// TwinCAT 3 PLC project FRANKA
// ProgramVersion: 3.1.4023.0
// libraries:
//   Tc2_Database, * (Beckhoff Automation GmbH)
//   Tc2_ModbusRTU, * (Beckhoff Automation GmbH)
//   Tc2_ModbusSrv, * (Beckhoff Automation GmbH)
//   Tc2_Standard, * (Beckhoff Automation GmbH)
//   Tc2_System, * (Beckhoff Automation GmbH)
//   Tc2_Utilities, * (Beckhoff Automation GmbH)
//   Tc3_Database, * (Beckhoff Automation GmbH)
//   Tc3_EventLogger, * (Beckhoff Automation GmbH)
//   Tc3_Module, * (Beckhoff Automation GmbH)
//   VisuSymbols,3.5.10.0,System
// project tree:
//   DUTs/ MS.TcTLEO, PLC_Data.TcDUT, ST_Table.TcDUT, DB_Columns.TcDUT, Visu_Data.TcDUT
//   / GlobalTextList.TcGTLO, PlcTask.TcTTO, Visualisierungsmanager.TcVMO (not stored)
//   GVLs/ GVL.TcGVL, GVL_IO.TcGVL, GVL_Persistent.TcGVL
//   POUs/ FB_Blinker.TcPOU, Initialize_Measurement_Values.TcPOU, MAIN.TcPOU, FB_NewTable.TcPOU, FB_DB_Write2.TcPOU, shutdown.TcPOU
//   VISUs/ Visualization.TcVIS
// real-time tasks:
//   TASK PlcTask: cycle T#10ms, priority 20, ADS port 350
//   TASK PlcTask1: cycle T#10ms, priority 21, ADS port 351
// I/O:
//   DEVICE Gerät 1 (EtherCAT Automation Protocol) (disabled), AmsNetId 192.168.26.100.2.1
//   DEVICE Gerät 3 (EtherCAT), AmsNetId 192.168.26.100.4.1
//     Klemme 1 (EK1100) [EK1100 EtherCAT-Koppler (2A E-Bus)]
//       Klemme 2 (EL2008) [EL2008 8K. Dig. Ausgang 24V, 0.5A]
//       Klemme 3 (EL2008) [EL2008 8K. Dig. Ausgang 24V, 0.5A]
//       Klemme 4 (EL1008) [EL1008 8K. Dig. Eingang 24V, 3ms]
//       Klemme 5 (EL2024) [EL2024 4K. Dig. Ausgang 24V, 2A]
//       Klemme 6 (EL9011) [EL9011 Endklemme]
// variable links:
//   FRANKA/FRANKA Instance <-> Device 3 (EtherCAT)/Term 1 (EK1100)/Term 2 (EL2008)
//     PlcTask Outputs/GVL.LED1 <-> Channel 4/Output
//     PlcTask Outputs/GVL.LED2 <-> Channel 1/Output
//     PlcTask Outputs/GVL.LED3 <-> Channel 7/Output
//     PlcTask Outputs/GVL.LED4 <-> Channel 6/Output
//     PlcTask Outputs/GVL.LED5 <-> Channel 8/Output
//     PlcTask Outputs/GVL.LED6 <-> Channel 3/Output
//     PlcTask Outputs/GVL.LED7 <-> Channel 5/Output
//     PlcTask Outputs/GVL.LED8 <-> Channel 2/Output
//   FRANKA/FRANKA Instance <-> Device 3 (EtherCAT)/Term 1 (EK1100)/Term 3 (EL2008)
//     PlcTask Outputs/GVL.Schalterlichtgrun <-> Channel 3/Output
//     PlcTask Outputs/GVL.Schalterlichtrot <-> Channel 1/Output
//     PlcTask Outputs/GVL.Schalterlichtweis <-> Channel 4/Output
//     PlcTask Outputs/GVL.schalterspannung <-> Channel 2/Output
//   FRANKA/FRANKA Instance <-> Device 3 (EtherCAT)/Term 1 (EK1100)/Term 4 (EL1008)
//     PlcTask Inputs/GVL.Grau_Schalter <-> Channel 1/Input
//     PlcTask Inputs/GVL.Start_Schalter <-> Channel 2/Input
//     PlcTask Inputs/GVL.Stop_Schalter <-> Channel 3/Input

CONFIGURATION FRANKA
    RESOURCE PLC ON TwinCAT3
        TASK PlcTask(INTERVAL := T#10ms, PRIORITY := 20);
        PROGRAM MAIN WITH PlcTask : MAIN;
    END_RESOURCE
END_CONFIGURATION

// ---- DUTs/MS.TcTLEO
{attribute 'qualified_only'}
{attribute 'strict'}
TYPE MS :
(
	Init_delay,
	Initialization,
	Start,
	Restart,
	NewTable_DB,
	Write_DB,
	FRANKA_Pick_and_place_PCB,
	FRANKA_Measure,
	LED_confirmation,
	FRANKA_Place_PCB,
	DB_Write,
	Measurement_counter,
	Reset,
	FRANKA_ERROR,
	measurebackup,
	Wait
	
);
END_TYPE

// ---- DUTs/PLC_Data.TcDUT
TYPE PLC_Data :
STRUCT
	PCB_ID			: 	INT;
	PCB_no_defects	:	STRING(50);
	Measurement_ID	: 	ARRAY [1..6] OF INT;
	TimeStamp		: 	ARRAY [1..6] OF DT;
	MeasureInTol	: 	ARRAY [1..6] OF STRING(50);
	Measure_Type	: 	ARRAY [1..6] OF STRING(50);
	Measure_Result	: 	ARRAY [1..6] OF REAL;
	Measure_Reference: 	ARRAY [1..6] OF REAL;
	Measure_Tolerance: 	ARRAY [1..6] OF REAL;

END_STRUCT
END_TYPE

// ---- DUTs/ST_Table.TcDUT
TYPE ST_Table :
STRUCT
sName: STRING(50);
sProperty: STRING;
nLength: UDINT;
eType: E_ColumnType;
END_STRUCT
END_TYPE

// ---- DUTs/DB_Columns.TcDUT
TYPE DB_Columns :
STRUCT
	PCB_Batch_ID: INT;
	PCB_ID: 		INT;
	Measurement_ID: INT;
	TimeStamp: 		DT;
	FreeFromDefects: STRING(50);
	Measure_Type: STRING(50);
	Measure_Result: REAL;
	Measure_Reference: REAL;
	Measure_Tolerance: REAL;	
END_STRUCT
END_TYPE

// ---- DUTs/Visu_Data.TcDUT
TYPE Visu_Data :
STRUCT
	PCB_Batch_ID	: 		INT;	
	PCB_ID			: 		INT;
	PCB_no_defects	:		STRING(50);
	Measure1InTol	: 		STRING(50);
	Measure2InTol	: 		STRING(50);
	Measure3InTol	: 		STRING(50);		
END_STRUCT
END_TYPE

// ---- GVLs/GVL.TcGVL
 {attribute 'qualified_only'}
VAR_GLOBAL
//Preset before program
	pcb_n			: INT;
	measure_n 		: INT;
	pcb_max			: INT;
	measure_max		: INT;

// MS Access Table Setting	
	ActiveTable		: STRING;
	
	
// fill during program
    Data: DB_Columns; // Data for MS Access Database
	PLC_Data: ARRAY [1..8] OF PLC_Data;// Data Saved in PLC
	Visu_Data: ARRAY [1..8] OF Visu_Data; // Visu Data
	

// DB_Writting
	Writing_finished: BOOL;
	write_state: INT;
	
// I/O Configuration
	
	LED1	AT%Q*:	BOOL;
	LED2	AT%Q*:	BOOL;
	LED3	AT%Q*:	BOOL;
	LED4	AT%Q*:	BOOL;
	LED5	AT%Q*:	BOOL;
	LED6	AT%Q*:	BOOL;
	LED7	AT%Q*:	BOOL;
	LED8	AT%Q*:	BOOL;
	
	Schalterlichtrot 	AT%Q*:	BOOL;
	Schalterlichtweis 	AT%Q*:	BOOL;
	Schalterlichtgrun 	AT%Q*:	BOOL;
	schalterspannung 	AT%Q*:	BOOL;
	
	Start_Schalter	AT%I*:	BOOL;
	Stop_Schalter	AT%I*:	BOOL;
	Grau_Schalter	AT%I*:	BOOL;
	
// Modbus Variabeln
	mb_Input_Coils      : ARRAY [0..255] OF BOOL;
	mb_Output_Coils     : ARRAY [0..255] OF BOOL;
	mb_Input_Registers  : ARRAY [0..255] OF WORD;
	mb_Output_Registers : ARRAY [0..255] OF WORD;

// Variables Measurement
	
sMeas_type	:	STRING;	// Measurement type first define measurement type then start
						// CSQ | CSD | CSR | CPQ | CPD | CPR | CPG | LSQ |LSD | LSR |
						// LPQ | LPD | LPR | LPG | ZTH | YTH | RX | GB | DCR |
bMeas_start	:	BOOL;	// start mearuement
rMeas_01	: 	REAL;	// Measurement result 1
rMeas_02	: 	REAL;	// Measurement result 2
bMeas_ready	:	BOOL;	// Measurement finished
bMeas_error	:	BOOL;	// Error flag
sMeas_errormsg:	STRING;	// Error Message String
bkill_proc	:	BOOL;	// Terminate Python Script

// Blocky start

        bStartBlockly 	: BOOL 		:= TRUE;
		sDeskUsername	: STRING 	:='Benjamin';
		sDeskPassword	: STRING	:='Benjamin';

// Init Measurement settings
Measurement_Init : BOOL;


END_VAR

// ---- GVLs/GVL_IO.TcGVL
{attribute 'qualified_only'}
VAR_GLOBAL
	// FRANKA OUTPUT Coils
	
	FRANKA_Marker0			:	REFERENCE TO BOOL;
	FRANKA_home1			:	REFERENCE TO BOOL;
	PCB_Marker2				: 	REFERENCE TO BOOL;
	FRANKA_MPoint_reached3	:	REFERENCE TO BOOL;
	FRANKA_Measurement_finished4: REFERENCE TO BOOL;
	FRANKA_PCB_Picked5		:	REFERENCE TO BOOL;
	FRANKA_PCB_Placed6		:	REFERENCE TO BOOL;
	FRANKA_ready_to_start	:	REFERENCE TO BOOL;

	// FRANKA INPUT Coils
	PLC_Measure_Finished0	: 	REFERENCE TO BOOL;
	PLC_confirm_PCB_placement1: 	REFERENCE TO BOOL;
	PLC_Start_trigger		:	REFERENCE TO BOOL;
	
END_VAR

// ---- GVLs/GVL_Persistent.TcGVL
{attribute 'qualified_only'}
VAR_GLOBAL PERSISTENT
		PCB_Batch_ID			: INT;


END_VAR

// ---- POUs/MAIN.TcPOU
PROGRAM MAIN
VAR




state : MS;

NewTable 	: FB_NewTable;
WriteDB		: FB_DB_Write;



// current file time

		fbSystemTime    : GETSYSTEMTIME;
        timeAsFileTime  : T_FILETIME;
        timeAsDT        : DT;
// Measurement trigger
		trig			: BOOL;

		
// Run Python script for measurement stuff
		runpython		: BOOL:=TRUE;
		Start_py_script : NT_StartProcess;
		
// Run Blockly & FRANKA Desk

//        bStartscript 	: BOOL := TRUE;
        bBusy 			: BOOL := FALSE;
        Start_py_script1 : NT_StartProcess;
		
// IPC Shut Down
		shutdown	:shutdown; 
	
// LED confirmation counter
k: INT :=1;

// Blink Funktion
fbBlinker_grun		:	FB_Blinker;	
fbBlinker_rot		:	FB_Blinker;
fbBlinker_weis		:	FB_Blinker;
green_init			:	BOOL;

// Init_delay
   Delay_startup		: TON;
   Delay			: TON;
   Start_init		: BOOL:=FALSE;
   Delay_init		: BOOL;
   
	clear: INT;
END_VAR

fbSystemTime( timeLoDW =>timeAsFileTime.dwLowDateTime , timeHiDW =>timeAsFileTime.dwHighDateTime );
timeAsDT := FILETIME_TO_DT( timeAsFileTime );

GVL_IO.FRANKA_Marker0 				REF= GVL.mb_Output_Coils[0];
GVL_IO.FRANKA_home1	 				REF= GVL.mb_Output_Coils[1];
GVL_IO.PCB_Marker2	 				REF= GVL.mb_Output_Coils[2];
GVL_IO.FRANKA_MPoint_reached3		REF= GVL.mb_Output_Coils[3];
GVL_IO.FRANKA_Measurement_finished4	REF= GVL.mb_Output_Coils[4];
GVL_IO.FRANKA_PCB_Picked5			REF= GVL.mb_Output_Coils[5];
GVL_IO.FRANKA_PCB_Placed6			REF= GVL.mb_Output_Coils[6];
GVL_IO.FRANKA_ready_to_start		REF= GVL.mb_Output_Coils[7];
GVL_IO.PLC_Measure_Finished0		REF= GVL.mb_Input_Coils[0];
GVL_IO.PLC_confirm_PCB_placement1	REF= GVL.mb_Input_Coils[1];
GVL_IO.PLC_Start_trigger			REF= GVL.mb_Input_Coils[2];

shutdown(Trig:=GVL.Grau_Schalter);
IF GVL.Stop_Schalter=TRUE THEN
	state:=MS.Reset;
END_IF


GVL.Data.PCB_Batch_ID:= GVL_Persistent.PCB_Batch_ID;




CASE state OF


MS.Reset : 	
			// Reset HMI
				IF clear<9 THEN
					GVL.Visu_Data[clear].PCB_Batch_ID:=0;
					GVL.Visu_Data[clear].PCB_ID:=0;
					GVL.Visu_Data[clear].PCB_no_defects:='';
					GVL.Visu_Data[clear].Measure1InTol:='';
					GVL.Visu_Data[clear].Measure2InTol:='';
					GVL.Visu_Data[clear].Measure3InTol:='';
					GVL.PLC_Data[clear].MeasureInTol[1]:='';
					GVL.PLC_Data[clear].MeasureInTol[2]:='';
					GVL.PLC_Data[clear].MeasureInTol[3]:='';					
					clear:=clear+1;
				END_IF

			
			// LEDs off
				GVL.LED1:=FALSE;
				GVL.LED2:=FALSE;
				GVL.LED3:=FALSE;
				GVL.LED4:=FALSE;
				GVL.LED5:=FALSE;
				GVL.LED6:=FALSE;
				GVL.LED7:=FALSE;
				GVL.LED8:=FALSE;
			//
            fbBlinker_weis(bStart:=TRUE , tPeriode:= T#1S, bBlinker=>GVL.Schalterlichtweis);
			GVL.Schalterlichtgrun:=FALSE;
			GVL.bStartBlockly := FALSE;
			GVL.measure_n:=1;
			GVL.pcb_n:=1;
			Start_init:=FALSE;
			GVL_IO.FRANKA_ready_to_start:=FALSE;
			Delay(IN:=FALSE);
			IF GVL.Grau_Schalter=TRUE THEN
				state:= MS.Start;
				// Batch ID Increment
				GVL_Persistent.PCB_Batch_ID:=GVL_Persistent.PCB_Batch_ID+1;
			END_IF
			
MS.Init_delay:
				Delay_startup(IN:=TRUE, PT:= T#10S, Q=>Start_init, ET=>);
				IF Start_init=TRUE THEN
					Start_init:=FALSE;
					state:=MS.Initialization;
				END_IF

MS.Initialization:

			// LEDs off
				GVL.LED1:=FALSE;
				GVL.LED2:=FALSE;
				GVL.LED3:=FALSE;
				GVL.LED4:=FALSE;
				GVL.LED5:=FALSE;
				GVL.LED6:=FALSE;
				GVL.LED7:=FALSE;
				GVL.LED8:=FALSE;
				

				GVL.Schalterlichtweis:=TRUE;
				GVL.schalterspannung:= TRUE;
			// Initialize Blockly & FRANKA Desk
					
			    IF GVL.bStartBlockly = TRUE AND bBusy = FALSE THEN
        			Start_py_script1(
            		NETID := '',
            		PATHSTR := 'blocklenium',
            		DIRNAME := 'C:\Users\Administrator\Desktop',
     				COMNDLINE := '--insecure-con --login-required -b PCB_Measure.url -u http://192.168.2.2/desk/',
					//COMNDLINE := '--insecure-con --login-required -b PCB_Handling.url -u http://192.168.2.2/desk/',
                	START := TRUE,
            		BUSY => bBusy
        			);
       			 	GVL.bStartBlockly := FALSE;
					//bBusy:= FALSE;
    			END_IF
			
				
				
		// Initialize Measurement script
		
			IF runpython = TRUE THEN	
				Start_py_script(NETID:='',
				PATHSTR:= 'bkpads',
				DIRNAME:= 'C:\Users\Administrator\Desktop\',
				COMNDLINE:='-c COM4',
				Start:=TRUE,
				TMOUT:=T#1S);
				runpython:=FALSE;
			 END_IF		
		

//			IF runpython = TRUE THEN	
//				Start_py_script(NETID:='',
//				PATHSTR:= 'C:\Python38\python.exe',
//				DIRNAME:= 'C:\Users\Administrator\Desktop\',
//				COMNDLINE:='C:\Users\Administrator\Desktop\bkpads.py',
//				Start:=TRUE,
//				TMOUT:=T#1S);
//				runpython:=FALSE;
//			 END_IF
			
			// Initializes, settings for measurement
			GVL.pcb_n:=1;
			GVL.pcb_max:=8;
			GVL.measure_n:=1;
			GVL.measure_max:=3;
			Initialize_Measurement_Values(); // Set Measurement references, tolerances & Types for measurement points on PCB
			
			IF GVL.Measurement_Init=TRUE THEN
			Delay_init:=TRUE;
			// Batch ID Increment
			GVL_Persistent.PCB_Batch_ID:=GVL_Persistent.PCB_Batch_ID+1;
			state:=MS.Start;
			;
			END_IF
			
			// Initialize table
			GVL.ActiveTable:='PCB_Test_Results';
			NewTable ();

MS.Restart:

			//
			GVL.Schalterlichtgrun:=FALSE;
			GVL.bStartBlockly := FALSE;
			GVL.measure_n:=1;
			GVL.pcb_n:=1;
			Start_init:=FALSE;
			Delay(IN:=FALSE);
			fbBlinker_grun(bStart:=Start_init , tPeriode:= T#1S, bBlinker=>GVL.Schalterlichtgrun);
			IF GVL.Start_Schalter= TRUE THEN			
				GVL.LED1:=FALSE;
				GVL.LED2:=FALSE;
				GVL.LED3:=FALSE;
				GVL.LED4:=FALSE;
				GVL.LED5:=FALSE;
				GVL.LED6:=FALSE;
				GVL.LED7:=FALSE;
				GVL.LED8:=FALSE;
				state:=MS.Start;		
			END_IF
					
			
			
			
			
			
MS.Start :	
			clear:=1;
			GVL.bStartBlockly := TRUE;
			Delay(IN:=Delay_init, PT:= T#30S, Q=>Start_init);
			
			IF Start_init = TRUE AND GVL_IO.FRANKA_ready_to_start=FALSE THEN
				state:= MS.FRANKA_ERROR;
			END_IF
			
		    fbBlinker_grun(bStart:=Start_init , tPeriode:= T#1S, bBlinker=>GVL.Schalterlichtgrun);
			
			
			GVL.Schalterlichtrot:=TRUE;
			IF GVL.Start_Schalter= TRUE THEN
				GVL_IO.PLC_Start_trigger:= TRUE;
			END_IF
			
			
			IF GVL_IO.FRANKA_Marker0 = TRUE THEN 
				GVL.Schalterlichtweis:= FALSE;
				GVL_IO.PLC_Start_trigger:= FALSE;
				fbBlinker_grun(bStart:=FALSE);
				state:=MS.FRANKA_Pick_and_place_PCB;
			ELSE ;
			END_IF
					
				
MS.FRANKA_Pick_and_place_PCB:

				IF GVL.pcb_n<=GVL.pcb_max THEN
					IF GVL_IO.FRANKA_PCB_Picked5 = TRUE THEN
						GVL_IO.PLC_confirm_PCB_placement1:=FALSE;
						state:=MS.FRANKA_Measure;
					END_IF
					ELSE;
						// finish program and write report from database
						state:=MS.Restart;
				END_IF
				
MS.FRANKA_Measure: 			
				IF GVL_IO.FRANKA_Measurement_finished4 = FALSE AND GVL_IO.FRANKA_MPoint_reached3 = TRUE THEN					
						GVL.sMeas_type:=GVL.PLC_Data[GVL.pcb_n].Measure_Type[GVL.measure_n];	// set type  
						IF  trig=FALSE THEN
							GVL.bMeas_start:= TRUE; // Trigger Measurement
							GVL_IO.PLC_Measure_Finished0:= FALSE;
							trig:=TRUE;
						END_IF
						IF GVL.bMeas_ready =TRUE THEN
							GVL.PLC_Data[GVL.pcb_n].Measure_Result[GVL.measure_n]:=GVL.rMeas_01;
							//rMeas_02	: 	REAL;	// Measurement result 2
							IF GVL.PLC_Data[GVL.pcb_n].Measure_Result[GVL.measure_n]<(GVL.PLC_Data[GVL.pcb_n].Measure_Reference[GVL.measure_n]+GVL.PLC_Data[GVL.pcb_n].Measure_Tolerance[GVL.measure_n]) AND GVL.PLC_Data[GVL.pcb_n].Measure_Result[GVL.measure_n]>(GVL.PLC_Data[GVL.pcb_n].Measure_Reference[GVL.measure_n]-GVL.PLC_Data[GVL.pcb_n].Measure_Tolerance[GVL.measure_n]) THEN
								GVL.PLC_Data[GVL.pcb_n].MeasureInTol[GVL.measure_n]:= 'Yes';

								ELSE
								GVL.PLC_Data[GVL.pcb_n].MeasureInTol[GVL.measure_n]:= 'No'; // test LED's YES otherwise No
								GVL.PLC_Data[GVL.pcb_n].PCB_no_defects:= 'defect';
								GVL.Visu_Data[GVL.pcb_n].PCB_no_defects:='defect';
							END_IF
							
							GVL_IO.PLC_Measure_Finished0:= TRUE;							
							IF GVL_IO.FRANKA_Marker0 =TRUE THEN
								state:=MS.DB_Write;
							END_IF
						END_IF
				END_IF

		
MS.DB_Write:
		// Visu Data
		GVL.Visu_Data[GVL.pcb_n].PCB_Batch_ID:=GVL_Persistent.PCB_Batch_ID;
		GVL.Visu_Data[GVL.pcb_n].PCB_ID:=GVL.pcb_n;
		GVL.Visu_Data[GVL.pcb_n].Measure1InTol:=GVL.PLC_Data[GVL.pcb_n].MeasureInTol[1];
		GVL.Visu_Data[GVL.pcb_n].Measure2InTol:=GVL.PLC_Data[GVL.pcb_n].MeasureInTol[2];
		GVL.Visu_Data[GVL.pcb_n].Measure3InTol:=GVL.PLC_Data[GVL.pcb_n].MeasureInTol[3];
		

		GVL.Data.PCB_ID:=GVL.pcb_n;
		GVL.Data.Measurement_ID:=GVL.measure_n;
		GVL.Data.Measure_Type:=GVL.PLC_Data[GVL.pcb_n].Measure_Type[GVL.measure_n];
		GVL.Data.TimeStamp:= timeASDT;
		GVL.Data.FreeFromDefects:=GVL.PLC_Data[GVL.pcb_n].MeasureInTol[GVL.measure_n];
		GVL.Data.Measure_Type:= GVL.PLC_Data[GVL.pcb_n].Measure_Type[GVL.measure_n];
		GVL.Data.Measure_Result:= GVL.PLC_Data[GVL.pcb_n].Measure_Result[GVL.measure_n];
		GVL.Data.Measure_Reference:= GVL.PLC_Data[GVL.pcb_n].Measure_Reference[GVL.measure_n];
		GVL.Data.Measure_Tolerance:= GVL.PLC_Data[GVL.pcb_n].Measure_Tolerance[GVL.measure_n];
		WriteDB ();
		IF GVL.Writing_finished=TRUE THEN
			GVL.write_state:=0;
			GVL_IO.FRANKA_MPoint_reached3:=FALSE;
			GVL.measure_n:=GVL.measure_n+1;
			trig:=FALSE;
			GVL.bMeas_ready:=FALSE;
		END_IF
																
		IF GVL.measure_n=GVL.measure_max+1 AND GVL.Writing_finished=TRUE THEN
			GVL_IO.PLC_Measure_Finished0:= FALSE;
			GVL.measure_n:=1;
			state:=MS.FRANKA_Place_PCB;	
			ELSE
			state:=MS.FRANKA_Measure;
		END_IF

				
							
MS.FRANKA_Place_PCB:
				
						IF GVL_IO.FRANKA_PCB_Placed6 = TRUE THEN
							
							GVL_IO.PLC_confirm_PCB_placement1:=TRUE;
							state:=MS.LED_confirmation;
							GVL_IO.FRANKA_PCB_Placed6:= FALSE;
						END_IF

MS.LED_confirmation:			
				// No defects in PCB?
				IF k<=GVL.measure_max THEN
					IF GVL.PLC_Data[GVL.pcb_n].MeasureInTol[k]='No' THEN
						GVL.pcb_n:=GVL.pcb_n+1;
						k:=1;
						state:=MS.FRANKA_Pick_and_place_PCB;			
					ELSE
						IF k=GVL.measure_max AND GVL.PLC_Data[GVL.pcb_n].MeasureInTol[k]='No' THEN
							GVL.pcb_n:=GVL.pcb_n+1;
							state:=MS.FRANKA_Pick_and_place_PCB;
							ELSE
							k:=k+1;
						END_IF
					END_IF
				ELSE
					CASE GVL.pcb_n OF
						1: GVL.LED1:=TRUE;
						   GVL.Visu_Data[1].PCB_no_defects:='Yes';
						2: GVL.LED2:=TRUE;
						   GVL.Visu_Data[2].PCB_no_defects:='Yes';
						3: GVL.LED3:=TRUE;
						   GVL.Visu_Data[3].PCB_no_defects:='Yes';
						4: GVL.LED4:=TRUE;
						   GVL.Visu_Data[4].PCB_no_defects:='Yes';
						5: GVL.LED5:=TRUE;
						   GVL.Visu_Data[5].PCB_no_defects:='Yes';
						6: GVL.LED6:=TRUE;
						   GVL.Visu_Data[6].PCB_no_defects:='Yes';
						7: GVL.LED7:=TRUE;
						   GVL.Visu_Data[7].PCB_no_defects:='Yes';
						8: GVL.LED8:=TRUE;
						   GVL.Visu_Data[8].PCB_no_defects:='Yes';
					END_CASE
						GVL.pcb_n:=GVL.pcb_n+1;
						k:=1;
						state:=MS.FRANKA_Pick_and_place_PCB;	
				END_IF	

	
MS.FRANKA_ERROR:
fbBlinker_rot(bStart:=TRUE , tPeriode:= T#0.2S, bBlinker=>GVL.Schalterlichtrot);
fbBlinker_grun(bStart:=TRUE , tPeriode:= T#1S, bBlinker=>GVL.Schalterlichtgrun);
fbBlinker_weis(bStart:=TRUE , tPeriode:= T#1S, bBlinker=>GVL.Schalterlichtweis);

MS.measurebackup:
				IF GVL_IO.FRANKA_Measurement_finished4 = FALSE AND GVL_IO.FRANKA_MPoint_reached3 = TRUE THEN					
						GVL.sMeas_type:=GVL.PLC_Data[GVL.pcb_n].Measure_Type[GVL.measure_n];	// set type  
						IF  trig=FALSE THEN
							GVL.bMeas_start:= TRUE; // Trigger Measurement
							GVL_IO.PLC_Measure_Finished0:= FALSE;
							trig:=TRUE;
						END_IF
						IF GVL.bMeas_ready =TRUE THEN
							GVL.PLC_Data[GVL.pcb_n].Measure_Result[GVL.measure_n]:=GVL.rMeas_01;
							//rMeas_02	: 	REAL;	// Measurement result 2
							IF GVL.PLC_Data[GVL.pcb_n].Measure_Result[GVL.measure_n]<(GVL.PLC_Data[GVL.pcb_n].Measure_Reference[GVL.measure_n]+GVL.PLC_Data[GVL.pcb_n].Measure_Tolerance[GVL.measure_n]) AND GVL.PLC_Data[GVL.pcb_n].Measure_Result[GVL.measure_n]>(GVL.PLC_Data[GVL.pcb_n].Measure_Reference[GVL.measure_n]-GVL.PLC_Data[GVL.pcb_n].Measure_Tolerance[GVL.measure_n]) THEN
								GVL.PLC_Data[GVL.pcb_n].MeasureInTol[GVL.measure_n]:= 'Yes';

								ELSE
								GVL.PLC_Data[GVL.pcb_n].MeasureInTol[GVL.measure_n]:= 'No'; // test LED's YES otherwise No
								GVL.PLC_Data[GVL.pcb_n].PCB_no_defects:= 'defect';
							END_IF
							
							GVL_IO.PLC_Measure_Finished0:= TRUE;
							
							
							IF GVL_IO.FRANKA_Marker0 =TRUE THEN
								GVL_IO.FRANKA_MPoint_reached3:=FALSE;
								GVL.measure_n:=GVL.measure_n+1;
								trig:=FALSE;
								GVL.bMeas_ready:=FALSE;
								
								
								IF GVL.measure_n=GVL.measure_max+1 THEN
									GVL_IO.PLC_Measure_Finished0:= FALSE;
									GVL.measure_n:=1;
									//state:=MS.FRANKA_Place_PCB;
									state:=MS.FRANKA_Place_PCB;	
								END_IF
							END_IF
						END_IF
				END_IF


				
				
//DB Write Backup
				GVL.Data.PCB_ID:=GVL.pcb_n;
				GVL.Data.Measurement_ID:=GVL.measure_n;
				GVL.Data.Measure_Type:=GVL.PLC_Data[GVL.pcb_n].Measure_Type[GVL.measure_n];
				GVL.Data.TimeStamp:= timeASDT;
				GVL.Data.FreeFromDefects:='Yes';
				GVL.Data.Measure_Type:= 'Resistance';
				GVL.Data.Measure_Result:= 43.3;
				GVL.Data.Measure_Reference:= 4.4;
				GVL.Data.Measure_Tolerance:= 0.2;
				WriteDB ();
				IF GVL.Writing_finished=TRUE THEN
				GVL.write_state:=0;
				END_IF

END_CASE

END_PROGRAM

// ---- POUs/FB_NewTable.TcPOU
FUNCTION_BLOCK FB_NewTable
VAR_INPUT
END_VAR
VAR_OUTPUT
END_VAR
VAR

fbPLCDBCreate : FB_PLCDBCreate(sNetID := '', tTimeout := T#5S);
ColumnInfo : ARRAY [0..8] OF ST_Table; // Worked with 0....7, before persistent
MAX_DBCOLUMNS : UDINT := 255;

END_VAR

//Column settings
ColumnInfo[0].sName := 'PCB_Batch_ID'; 		ColumnInfo[0].eType := E_ColumnType.Integer; 	ColumnInfo[0].nLength := 4; ColumnInfo[0].sProperty := 'IDENTITY(1,1)';
ColumnInfo[1].sName := 'PCB_ID'; 			ColumnInfo[1].eType := E_ColumnType.Integer; 	ColumnInfo[1].nLength := 4;
ColumnInfo[2].sName := 'Measurement_ID'; 	ColumnInfo[2].eType := E_ColumnType.Integer; 	ColumnInfo[2].nLength := 4;
ColumnInfo[3].sName := 'TimeStamp'; 		ColumnInfo[3].eType := E_ColumnType.DateTime; 	ColumnInfo[3].nLength := 4;
ColumnInfo[4].sName := 'FreeFromDefects'; 	ColumnInfo[4].eType := E_ColumnType.NVarChar; 	ColumnInfo[4].nLength := 50;
ColumnInfo[5].sName := 'Measure_Type'; 		ColumnInfo[5].eType := E_ColumnType.NVarChar; 	ColumnInfo[5].nLength := 50;
ColumnInfo[6].sName := 'Measure_Result'; 	ColumnInfo[6].eType := E_ColumnType.REAL_; 		ColumnInfo[6].nLength := 4;
ColumnInfo[7].sName := 'Measure_Reference'; ColumnInfo[7].eType := E_ColumnType.REAL_; 		ColumnInfo[7].nLength := 4;
ColumnInfo[8].sName := 'Measure_Tolerance'; ColumnInfo[8].eType := E_ColumnType.REAL_; 		ColumnInfo[8].nLength := 4;




fbPLCDBCreate.Table(
hDBID:= 1, 
sTableName:= GVL.ActiveTable, 
pTableCfg:= ADR(ColumnInfo), 
cbTableCfg:= SIZEOF(ColumnInfo));

END_FUNCTION_BLOCK

// ---- POUs/FB_DB_Write2.TcPOU
FUNCTION_BLOCK FB_DB_Write
VAR_INPUT
END_VAR
VAR_OUTPUT
END_VAR
VAR

//DB Write variables 1..8 without persistent
stTable_structure: DB_Columns;
fbPLCDBWrite	: FB_PLCDBWrite(sNetID:='', tTimeout:=T#5S);
arrColumns: ARRAY [1..9] OF STRING (50) := [
'PCB_Batch_ID',
'PCB_ID',
'Measurement_ID',
'TimeStamp',
'FreeFromDefects',
'Measure_Type',
'Measure_Result',
'Measure_Reference',
'Measure_Tolerance'];
ipTcResult: I_TcResultEvent;

//DB Read variables
fbPLCDBRead: FB_PLCDBRead(sNetID:='', tTimeout:=T#5S);
arrRecords: ARRAY [1..8] OF DB_Columns;

// case 200
			sSourcePath:  STRING(255);
			sEventClasse :  WSTRING(255);
			nEventID:  E_Severity;
			nEventText :  WSTRING(255);

// Current time





END_VAR


// e_nums //elemente mit Namen ansprechen. 
CASE GVL.write_state OF

0: // IDl

GVL.Writing_finished:= FALSE;
GVL.write_state:=1;
	;
1:  //Write
	fbPLCDBWrite.WriteStruct(
		hDBID:= 1,
		sTableName:= GVL.ActiveTable,
		pRecord:= ADR(GVL.Data),
		cbRecord:= SIZEOF (GVL.Data),		
		pColumnNames:= ADR(arrColumns),
		cbColumnNames:=SIZEOF(arrColumns));

		IF NOT fbPLCDBWrite.bBusy THEN
		ipTcResult:= fbPLCDBWrite.ipTcResultEvent;
			IF NOT fbPLCDBWrite.bError THEN
				GVL.write_state:=2;
			ELSE
				GVL.write_state:= 200;
			END_IF
		END_IF

2:
	fbPLCDBRead.ReadStruct(
		hDBID:= 1, 
		sTableName:= GVL.ActiveTable, 
		pColumnNames:= ADR(arrColumns), 
		cbColumnNames:= SIZEOF(arrColumns), 
		sOrderByColumn:= 'ID', 
		eOrderType:= E_OrderType.ASC, 
		nStartIndex:= 0, 
		nRecordCount:= 8, 
		pData:= ADR(arrRecords), 
		cbData:=SIZEOF (arrRecords));			
		IF NOT fbPLCDBRead.bBusy THEN
			ipTcResult:= fbPLCDBRead.ipTcResultEvent;
			IF NOT fbPLCDBRead.bError THEN
				GVL.write_state:=200;
			ELSE
				GVL.write_state:= 200;
			END_IF
		END_IF

200: 	sSourcePath:=ipTcResult.SourcePath;
		sEventClasse := ipTcResult.EventClassDisplayName;
		nEventID:= ipTcresult.Severity;
		nEventText := ipTcResult.Text;
		GVL.write_state:=3;
		
3: 		GVL.Writing_finished:=TRUE;
END_CASE

END_FUNCTION_BLOCK

// ---- POUs/shutdown.TcPOU
FUNCTION_BLOCK shutdown
VAR_INPUT
	Trig: BOOL;
	Shut: NT_Shutdown;
END_VAR
VAR_OUTPUT
END_VAR
VAR
	Timer: TON;
	Shutd:NT_Shutdown;
END_VAR

Timer(IN := Trig, PT := T#5s); // TON
Shut(DELAY := 10, START := Timer.Q); // NT_Shutdown

END_FUNCTION_BLOCK

// ---- POUs/FB_Blinker.TcPOU
FUNCTION_BLOCK FB_Blinker
VAR_INPUT
		bStart		:	BOOL;
	    tPeriode	:	TIME	:= T#1S;
END_VAR
VAR_OUTPUT
		bBlinker	: 	BOOL;
END_VAR
VAR
		fbTimer 	: 	TON;
END_VAR

fbTimer (IN:=bStart AND NOT fbTimer.Q, PT:= tPeriode,);

IF fbTimer.ET >= tPeriode/2
	THEN
	bBlinker:= TRUE;
	ELSE
	bBlinker:=FALSE;
	
END_IF

END_FUNCTION_BLOCK

// ---- POUs/Initialize_Measurement_Values.TcPOU
PROGRAM Initialize_Measurement_Values
VAR
	n : INT:=1;
	c : INT;

END_VAR

// Setting PCB
// Measurement Types 
// CSQ | CSD | CSR | CPQ | CPD | CPR | CPG | LSQ |LSD | LSR |
// LPQ | LPD | LPR | LPG | ZTH | YTH | RX | GB | DCR |
IF n<9 THEN
	// Setting Measurement Point 1 Resistance1
	c:=1;
	GVL.PLC_Data[n].Measure_Type[c] 		:='RX';
	GVL.PLC_Data[n].Measure_Reference[c]	:=680;
	GVL.PLC_Data[n].Measure_Tolerance[c]	:=34;
	// Setting Measurement Point 2 Capacitance1
	c:=2;
	GVL.PLC_Data[n].Measure_Type[c] 		:='CSQ';
	GVL.PLC_Data[n].Measure_Reference[c]	:=2.2E-08;
	GVL.PLC_Data[n].Measure_Tolerance[c]	:=2.2E-09;
	// Setting Measurement Point 3 Resistance2
	c:=3;
	GVL.PLC_Data[n].Measure_Type[c] 		:='RX';
	GVL.PLC_Data[n].Measure_Reference[c]	:=680;
	GVL.PLC_Data[n].Measure_Tolerance[c]	:=34;
		// Setting Measurement Point 3 Inductor 2
	c:=4;
	GVL.PLC_Data[n].Measure_Type[c] 		:='LPD';
	GVL.PLC_Data[n].Measure_Reference[c]	:=5;
	GVL.PLC_Data[n].Measure_Tolerance[c]	:=10;
		// Setting Measurement Point 3 Resistor 1
	c:=5;
	GVL.PLC_Data[n].Measure_Type[c] 		:='LPD';
	GVL.PLC_Data[n].Measure_Reference[c]	:=5;
	GVL.PLC_Data[n].Measure_Tolerance[c]	:=10;
		// Setting Measurement Point 3 Resistor 2
	c:=6;
	GVL.PLC_Data[n].Measure_Type[c] 		:='LPD';
	GVL.PLC_Data[n].Measure_Reference[c]	:=5;
	GVL.PLC_Data[n].Measure_Tolerance[c]	:=10;


    n:=n+1;

IF n=9 THEN
	GVL.Measurement_Init:= TRUE;
END_IF

END_IF

END_PROGRAM

// ---- VISUs/Visualization.TcVIS
VISUALIZATION Visualization  // 2x2
END_VISUALIZATION
